// TIA Portal V17 export
// export: Created 2023-02-13T11:15:57.9574922Z, ExportSetting WithDefaults, DisplayName Totally Integrated Automation Portal, DisplayVersion V17, DisplayName TIA Portal Openness, DisplayVersion V17, DisplayName TIA Portal Teamcenter Gateway, DisplayVersion V17, DisplayName TIA Portal Version Control Interface, DisplayVersion V17, DisplayName SINAMICS Startdrive Advanced, DisplayVersion V17, DisplayName SINAMICS Startdrive G130, G150, S120, S150, SINAMICS MV, S210, DisplayVersion V17, DisplayName SINAMICS Startdrive G110M, G120, G120C, G120D, G120P, G115D, DisplayVersion V17, DisplayName STEP 7 Professional, DisplayVersion V17, DisplayName STEP 7 Safety, DisplayVersion V17, DisplayName WinCC Professional, DisplayVersion V17
FUNCTION_BLOCK "Danfos_VSD"   // FB623, LAD
{ S7_Optimized_Access := 'FALSE' }
VERSION : 0.1
// stored: AutoNumber false, IsIECCheckEnabled false, SetENOAutomatically false, UDAEnableTagReadback false
   VAR_INPUT
      In_CMD : Bool;   // 0 = Stop, 1 = Start
      Reset : Bool;
      QuickStop : Bool;   // 1 = Emergency stop
      drive_f_setpoint : Real;   // Frequency setpoint in Hz; 0.00<f_setl<50.00Hz
      In_STW : Word;
      drive_AV { ExternalAccessible := 'False'; ExternalVisible := 'False'; ExternalWritable := 'False'} : Int;   // Drive Actual value
   END_VAR
   VAR_OUTPUT
      Danfos_CTW : Word;
      Danfos_SP { ExternalAccessible := 'False'; ExternalVisible := 'False'; ExternalWritable := 'False'} : Word;   // Drive Settpoint
      Drive_OK : Bool;
      Drive_Run : Bool;
      QAlarm : Word;
      Danfos_f_act : Real;   // actual_frequency 0...50Hz
      "Danfos_QAV_%" : Real;   // actual_frequency 0..100%
   END_VAR
   VAR DB_SPECIFIC
      SW : Struct
         "Bit 0-Control" : Bool;   // 0 = Control not ready, 1 = Control ready
         "Bit 1-Drive" : Bool;   // 0 = Drive not ready, 1 = Drive ready
         "Bit 2-Coasting stop" : Bool;   // 0 = can't start the motor, 1 = can start the motor
         "Bit 3-Trip" : Bool;   // 0 = No error, 1 = Trip
         "Bit 4-Error" : Bool;   // 0 = No error, 1 = Drive Error (no Trip)
         "Bit 5-NOP" : Bool;
         "Bit 6-triplock" : Bool;   // 0 = not in fault, 1 = tripped and locked
         "Bit 7-Warning" : Bool;   // 0 = No warning , 1 = Warning
         "Bit 8-Speed reference" : Bool;   // 0 = Speed =/ reference, 1 = Speed = reference
         "Bit 9-Operation" : Bool;   // 0 = Local operation, 1 = bus control
         "Bit 10-frequency range" : Bool;   // 0 = Outside frequency range, 1 =Within frequency range
         "Bit 11-Operation" : Bool;   // 0 = No operation, 1 = In operation
         "Bit 12-Drive OK" : Bool;   // 0 = Drive OK, 1 = Stopped, autostart
         "Bit 13-Voltage OK" : Bool;   // 0 = Voltage OK, 1 = Voltage exceeded
         "Bit 14-Torque OK" : Bool;   // 0 = Torque OK, 1 = Torque exceeded
         "Bit 15-Timers OK" : Bool;   // 0 = Timers OK, 1 = Timers exceeded
      END_STRUCT;
      Reset_PE : Bool;
      Reset_Bits : Bool;
      f_act : Real;
   END_VAR
   VAR_TEMP   // added for the SCL form of the ladder/FBD networks
      _w1 : Bool;
   END_VAR
BEGIN

REGION Network 1: Reset
   // Bit Bit value=0 Bit value=1
   // 00 Reference value External selection lsb
   // 01 Reference value External selection msb
   // 02 DC brake Ramp
   // 03 Coasting No coasting
   // 04 Quick stop Ramp
   // 05 Hold output frequency Use ramp
   // 06 Ramp stop Start
   // 07 No function Reset
   // 08 No function Jog
   // 09 Ramp 1 Ramp 2
   // 10 Data invalid Data valid
   // 11 No function Relay 01 active
   // 12 No function Relay 04 active
   // 13 Parameter set-up selection lsb
   // 14 Parameter set-up selection msb
   // 15 No function Reverse
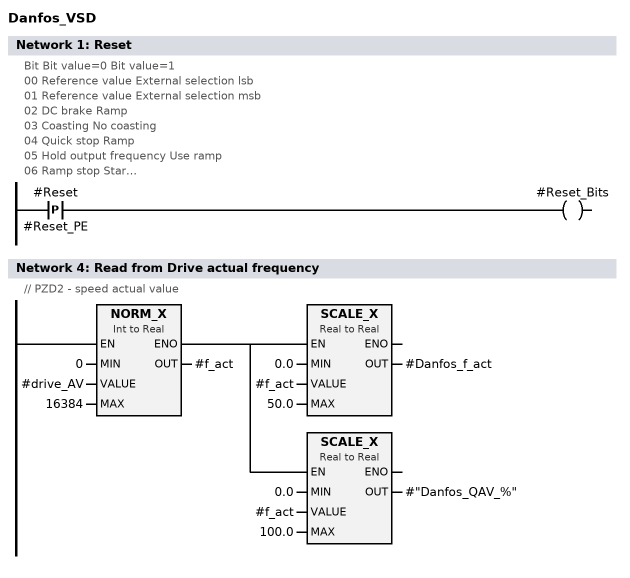
   RUNG wire#powerrail
      P_Contact(operand := #Reset, bit := #Reset_PE)
      Coil( #Reset_Bits )
   END_RUNG
   // the same network as SCL:
   #_w1 := #Reset AND NOT #Reset_PE;   // rising edge of #Reset
   #Reset_PE := #Reset;
   #Reset_Bits := #_w1;
END_REGION

REGION Network 2 (SCL): Read Status Word
   #SW."Bit 0-Control" := #In_STW.%X0;
   #SW."Bit 1-Drive" := #In_STW.%X1;
   #SW."Bit 2-Coasting stop" := #In_STW.%X2;
   #SW."Bit 3-Trip" := #In_STW.%X3;
   #SW."Bit 4-Error" := #In_STW.%X4;
   #SW."Bit 5-NOP" := #In_STW.%X5;
   #SW."Bit 6-triplock" := #In_STW.%X6;
   #SW."Bit 7-Warning" := #In_STW.%X7;
   #SW."Bit 8-Speed reference" := #In_STW.%X8;
   #SW."Bit 9-Operation" := #In_STW.%X9;
   #SW."Bit 10-frequency range" := #In_STW.%X10;
   #SW."Bit 11-Operation" := #In_STW.%X11;
   #SW."Bit 12-Drive OK" := #In_STW.%X12;
   #SW."Bit 13-Voltage OK" := #In_STW.%X13;
   #SW."Bit 14-Torque OK" := #In_STW.%X14;
   #SW."Bit 15-Timers OK" := #In_STW.%X15;
END_REGION

REGION Network 3 (SCL): Drive Status
   #Drive_Run := #SW."Bit 11-Operation" = true;

   #Drive_OK := (#SW."Bit 0-Control" = true AND
                 #SW."Bit 1-Drive" = true ) OR
                 (#SW."Bit 2-Coasting stop" = true AND
                 #SW."Bit 3-Trip" = false AND
                 #SW."Bit 4-Error" = false AND
                 #SW."Bit 6-triplock" = false AND
                 #SW."Bit 7-Warning" = false);
END_REGION

REGION Network 4: Read from Drive actual frequency
   // // PZD2 - speed actual value
   RUNG wire#powerrail
      { S7_Templates := "[SrcType := Int, DestType := Real]" } Normalize(min := 0, value := #drive_AV, max := 16384, out => #f_act)
      wire#w1
      { S7_Templates := "[SrcType := Real, DestType := Real]" } Scale(min := 0.0, value := #f_act, max := 50.0, out => #Danfos_f_act)
   END_RUNG
   RUNG wire#w1
      { S7_Templates := "[SrcType := Real, DestType := Real]" } Scale(min := 0.0, value := #f_act, max := 100.0, out => #"Danfos_QAV_%")
   END_RUNG
   // the same network as SCL:
   #f_act := NORM_X(MIN := 0, VALUE := #drive_AV, MAX := 16384);
   #Danfos_f_act := SCALE_X(MIN := 0.0, VALUE := #f_act, MAX := 50.0);
   #"Danfos_QAV_%" := SCALE_X(MIN := 0.0, VALUE := #f_act, MAX := 100.0);
END_REGION

REGION Network 5 (SCL): Write to Drive Control Word
   #Danfos_CTW.%X0 := false;
   #Danfos_CTW.%X1 := false;
   #Danfos_CTW.%X2 := true;
   #Danfos_CTW.%X3 := true;
   #Danfos_CTW.%X4 := #QuickStop = true;
   #Danfos_CTW.%X5 := true;
   #Danfos_CTW.%X6 := (#Drive_OK =true AND #In_CMD =true AND #QuickStop = true);
   #Danfos_CTW.%X7 := #Reset_Bits;
   #Danfos_CTW.%X8 := false;
   #Danfos_CTW.%X9 := false;
   #Danfos_CTW.%X10 := true;
   #Danfos_CTW.%X11 := false;
   #Danfos_CTW.%X12 := false;
   #Danfos_CTW.%X13 := false;
   #Danfos_CTW.%X14 := false;
   #Danfos_CTW.%X15 := false;
END_REGION

NETWORK
TITLE = Write to Drive Setpoint
// PZD2 - speed setpoint
// Valid speed setpoint between 0.00-50.00 Hz

      L     #drive_f_setpoint;  // Load the frequency setpoint [Hz]
      L     0.0;  // Load the value 0
      <R;  // Compare the speed setpoint with 0 (Hz): < 0 Hz ?
      JC    N004;  // Yes: Jump to mark N004; No: Continue program run

      L     #drive_f_setpoint;  // Load the frequency setpoint [Hz]
      L     50.0;  // Load the value 50
      >R;  // Compare the speed setpoint with 50 (Hz): > 50 Hz ?
      JC    N004;  // Yes: Jump to the mark N004; No: Continue program run

      L     #drive_f_setpoint;  // Load the frequency setpoint [Hz]

// Save 2 decimal places:
      L     100.0;  // Load the value 100
      *R;  // Multiply the values
      RND;  // Round-off the value (floating point number) to an integer number
      L     16384;  // Load the value 16384 = 4000HEX = 50Hz
      *D;  // Multiply the values
      L     5000;  // The load the value 5000
      /D;  // Divide the contents of AKKU2 by the contents of AKKU1
      T     #Danfos_SP;  // Transfer to the drive

N004: NOP   0;  // Jump mark N004: No function

END_FUNCTION_BLOCK
